(* CoDeSys 2.3 export: TRANSPORTSUBSTATUS.EXP *)

(* Data type in ENUM *)
TYPE TransportSubStatus : (TransportSubStatusNormal:=0, TransportSubStatusChangeSpeed, TransportSubStatusStarting, TransportSubStatusRefStopped,
								TransportSubStatusRefAlalrm, TransportSubStatusStopping, TransportSubStatusAlarm, TransportSubStatusTimeout,
								TransportSubStatusConfErr, TransportSubStatusUnknownCommand, TransportSubStatusBadCommandParameter);
END_TYPE
